KUKA KRL program: tipdress2.src, tipdress2.dat

--- tipdress2.src ---
&ACCESS RV1
&REL 33
&COMMENT TIPDRESS EXTERNAL GUN 2
DEF tipdress2( )
;================================================
; MODEL    :
; IE GROUP :
; STATION  :
; ROBOT    :
; FUNCTION : TIPDRESS EXTERNAL GUN 2
;================================================
;FOLD INI
;FOLD BASISTECH INI
GLOBAL INTERRUPT DECL 3 WHEN $STOPMESS==TRUE DO IR_STOPM ( )
INTERRUPT ON 3
BAS (#INITMOV,0 )
;ENDFOLD (BASISTECH INI)
;FOLD SPOTTECH INI
USERSPOT(#INIT)
;ENDFOLD (SPOTTECH INI)
;FOLD GRIPPERTECH INI
USER_GRP(0,DUMMY,DUMMY,GDEFAULT)
;ENDFOLD (GRIPPERTECH INI)
;FOLD USER INI
;Make your modifications here
;ENDFOLD (USER INI)
;ENDFOLD (INI)


pgno1_type=0

;FOLD PTP P10 H RETR OPN Gun= 2 Pair= FIRST Tool[14]:C520 Sin Pieza Base[0];%{PE}%R 6.1.2,%MKUKATPSPOT,%CRETR,%VPTP,%P 1:PTP, 2:P10, 3:, 5:100, 7:H, 9:#OPN, 11:2, 13:#FIRST
$BWDSTART=FALSE
PDAT_ACT=PH
FDAT_ACT=FP10
BAS(#PTP_PARAMS,PH.VEL)
S_ACT.GUN=2
S_ACT.PAIR=#FIRST
S_ACT.RETR=#OPN
S_READY=FALSE
TRIGGER WHEN DISTANCE=1 DELAY=0.0 DO USERSPOT(#RETR, S_ACT) PRIO=-1
PTP XP10
WAIT FOR S_READY
;ENDFOLD

;FOLD TDRESS.Swing_Forward 2 ;%{PE}%MKUKATPUSER
B_TDRESS=TDRESS (#SW_FWD ,2)
;ENDFOLD

;FOLD WAIT Time=1.5 sec;%{PE}%R 5.6.13,%MKUKATPBASIS,%CWAIT,%VWAIT,%P 2:1.5
WAIT SEC 1.5
;ENDFOLD

REPEAT

;FOLD TDRESS.Select_Active_Electrode 2 ;%{PE}%MKUKATPUSER
B_TDRESS=TDRESS (#TD_SEL ,2)
;ENDFOLD

pgno1_type=0
PGNO1=66

;FOLD TDRESS.Start_Cutter_Gun 2 ;%{PE}%MKUKATPUSER
B_TDRESS=TDRESS (#TD_START ,2)
;ENDFOLD

;FOLD TDRESS.Start_Count_Rotations 2 ;%{PE}%MKUKATPUSER
B_TDRESS=TDRESS (#CNT_STRT ,2)
;ENDFOLD

;FOLD CLOSE GUN 2 (3 TIMES) AND CHECK
$ADVANCE=0

FOR I=1 TO  3
CLOSEGUN (3 )

WAIT SEC 0.9



OPENGUN (3 )
ENDFOR
$ADVANCE=3
;endfold

;FOLD TDRESS.Stop_Count_Rotations 2 ;%{PE}%MKUKATPUSER
B_TDRESS=TDRESS (#CNT_STOP ,2)
;ENDFOLD

;FOLD TDRESS.Check_Rotations_Gun 2 Amount Of Rotations , 2 ;%{PE}%MKUKATPUSER
B_TDRESS=TDRESS (#CNT_CHK ,2, 2)
;ENDFOLD

UNTIL B_TDRESS==TRUE

;OPEN ARM OF THE DRESS

;FOLD TDRESS.Swing_Backward 2 ;%{PE}%MKUKATPUSER
B_TDRESS=TDRESS (#SW_BWD ,2)
;ENDFOLD

;FOLD TDRESS.Reset_Counter_Timer 2  Gun nr, 1 ;%{PE}%MKUKATPUSER
B_TDRESS=TDRESS (#TD_RES_CNT ,2, 1)
;ENDFOLD

;FOLD PTP Best_Praktisch H SPOT Gun= 2 Pair= FIRST RETR OPN INDEX1= 64 INDEX2= 1 Tool[14]:C520 Sin Pieza Base[0];%{PE}%R 6.1.2,%MKUKATPSPOT,%CSPOT,%VPTP,%P 1:PTP, 2:Best_Praktisch, 3:, 5:100, 7:H, 10:2, 12:#FIRST, 14:#OPN, 16:64, 18:1, 20:0, 22:0, 24:0, 25:SDAT3
$BWDSTART=FALSE
PDAT_ACT=PH
FDAT_ACT=FBest_Praktisch
BAS(#PTP_PARAMS,PH.VEL)
S_ACT.GUN=2
S_ACT.PAIR=#FIRST
S_ACT.RETR=#OPN
S_ACT.CLO_TM=SDEFAULT.CLO_TM
S_ACT.PGNO1=64
S_ACT.PGNO2=1
S_ACT.PRESS1=SDEFAULT.PRESS1
S_ACT.PRESS2=SDEFAULT.PRESS2
S_READY=FALSE
USERSPOT(#ADVSPOT, S_ACT)
TRIGGER WHEN DISTANCE=1 DELAY=SDEFAULT.CLO_TM DO USERSPOT(#PRESPOT, S_ACT) PRIO=-1
TRIGGER WHEN DISTANCE=1 DELAY=0.0 DO USERSPOT(#SPOT, S_ACT) PRIO=-1
PTP XBest_Praktisch
WAIT FOR S_READY
;ENDFOLD


END

;FOLD SETOUTPUT - SETS OUTPUT IF CONDITIONS ARE OK
DEF  SETOUTPUT (NR :IN,STATE :IN )
;************************************************************
;Function:  sets if to state value
;************************************************************
INT NR
BOOL STATE

IF (NR<>0) THEN
IF (NR>0) THEN
CONTINUE
$OUT[NR]=STATE
ELSE
CONTINUE
$OUT[-NR]= NOT STATE
ENDIF
ENDIF
END ;SetOutput
;ENDFOLD

;FOLD CHKINPUT - CHECKS INPUT <1 & RETURNS INPUT VALUE
DEFFCT  BOOL CHKINPUT(NR :IN,STATE :IN)
;************************************************************
;Function: checks if input nr<1 and returns input value
;************************************************************
INT NR
BOOL STATE

IF (NR<>0) THEN
IF (NR>0) THEN
RETURN  ($IN[NR]==STATE)
ELSE
RETURN  ($IN[-NR]==STATE)
ENDIF
ELSE
RETURN  (TRUE)
ENDIF
ENDFCT ; ChkInput
;ENDFOLD

;FOLD TIMEOUT - WAITS FOR CONDITION WITH TIMEOUT
DEFFCT  BOOL TIMEOUT(CONDITION :OUT,STATE :IN,MAXTIME :IN)
;************************************************************
;Function: waits for condition with timeout
;************************************************************
BOOL CONDITION
BOOL STATE
REAL MAXTIME

$TIMER[5]=-MAXTIME*1000
$TIMER_STOP[5]=FALSE
WHILE  (CONDITION<>STATE) AND  NOT ($TIMER_FLAG[5])
ENDWHILE
RETURN  ($TIMER_FLAG[5])
ENDFCT ; of TimeOut
;ENDFOLD

;FOLD CLOSEGUN - CLOSES WELDGUN BEFORE WELDING
DEF  CLOSEGUN (MYGUN :IN )
;************************************************************
;Function: closes and checks a gun
;************************************************************
INT MYGUN

SETOUTPUT (GRIPPER[MYGUN].OUT2,FALSE )
PULSE ($OUT[GRIPPER[MYGUN].OUT1],TRUE,0.2)
$TIMER[5]=-WAITTIME*1000
$TIMER_STOP[5]=FALSE
WHILE  ((CHKINPUT(GRIPPER[MYGUN].IN1,TRUE) AND CHKINPUT(GRIPPER[MYGUN].IN2,FALSE) AND CHKINPUT(GRIPPER[MYGUN].IN3,FALSE))<>TRUE) AND  NOT ($TIMER_FLAG[5])
ENDWHILE
IF ($TIMER_FLAG[5]) THEN
ERROR_DCP=TRUE
$MSG_T.RELEASE=FALSE
EMPTY_MSG={MSG_T: VALID FALSE,RELEASE FALSE,TYP #NOTIFY,MODUL[] " ",KEY[] " ",PARAM_TYP #VALUE,PARAM[] " ",DLG_FORMAT[] " ",ANSWER 0}
$MSG_T.TYP=#STATE
$MSG_T.KEY[]="Prestroke not closed        "
$MSG_T.VALID=TRUE
WAIT FOR  (($IN[GRIPPER[MYGUN].IN1]==TRUE) AND ($IN[GRIPPER[MYGUN].IN2]==FALSE) AND ($IN[GRIPPER[MYGUN].IN3]==FALSE))
$MSG_T.RELEASE=TRUE
WHILE $MSG_T.VALID
ENDWHILE
ERROR_DCP=FALSE
ENDIF

SETOUTPUT (GRIPPER[MYGUN].OUT3,TRUE )
SETOUTPUT (GRIPPER[MYGUN].OUT4,TRUE )
$TIMER[5]=-WAITTIME*1000
$TIMER_STOP[5]=FALSE
WHILE  ((CHKINPUT(GRIPPER[MYGUN].IN1,FALSE) AND CHKINPUT(GRIPPER[MYGUN].IN2,FALSE) AND CHKINPUT(GRIPPER[MYGUN].IN3,TRUE))<>TRUE) AND  NOT ($TIMER_FLAG[5])
ENDWHILE
IF ($TIMER_FLAG[5]) THEN
ERROR_DCP=TRUE
$MSG_T.RELEASE=FALSE
EMPTY_MSG={MSG_T: VALID FALSE,RELEASE FALSE,TYP #NOTIFY,MODUL[] " ",KEY[] " ",PARAM_TYP #VALUE,PARAM[] " ",DLG_FORMAT[] " ",ANSWER 0}
$MSG_T.TYP=#STATE
$MSG_T.KEY[]="Weldstroke not closed              "
$MSG_T.VALID=TRUE
WAIT FOR  (($IN[GRIPPER[MYGUN].IN1]==FALSE) AND ($IN[GRIPPER[MYGUN].IN2]==FALSE) AND ($IN[GRIPPER[MYGUN].IN3]==TRUE))
$MSG_T.RELEASE=TRUE
WHILE $MSG_T.VALID
ENDWHILE
ERROR_DCP=FALSE
ENDIF

END ;CLOSEGUN

;ENDFOLD

;FOLD OPENGUN - OPENS GUN FULLY AFTER WELDING
DEF  OPENGUN (MYGUN :IN )
;************************************************************
;Function: opens and checks a gun
;************************************************************
INT MYGUN
INT ANSWER

SETOUTPUT (GRIPPER[MYGUN].OUT3,FALSE )
SETOUTPUT (GRIPPER[MYGUN].OUT4,FALSE )
SETOUTPUT (GRIPPER[MYGUN].OUT1,FALSE )
PULSE ($OUT[GRIPPER[MYGUN].OUT2],TRUE,0.2)
$TIMER[5]=-WAITTIME*1000
$TIMER_STOP[5]=FALSE
WHILE  ((CHKINPUT(GRIPPER[MYGUN].IN1,FALSE) AND CHKINPUT(GRIPPER[MYGUN].IN2,TRUE) AND CHKINPUT(GRIPPER[MYGUN].IN3,FALSE))<>TRUE) AND  NOT ($TIMER_FLAG[5])
ENDWHILE
IF ($TIMER_FLAG[5]) THEN
ERROR_DCP=TRUE
$MSG_T.RELEASE=FALSE
EMPTY_MSG={MSG_T: VALID FALSE,RELEASE FALSE,TYP #NOTIFY,MODUL[] " ",KEY[] " ",PARAM_TYP #VALUE,PARAM[] " ",DLG_FORMAT[] " ",ANSWER 0}
$MSG_T.TYP=#STATE
$MSG_T.KEY[]="Prestroke not open                 "
$MSG_T.VALID=TRUE
WAIT FOR  (($IN[GRIPPER[MYGUN].IN1]==FALSE) AND ($IN[GRIPPER[MYGUN].IN2]==TRUE) AND ($IN[GRIPPER[MYGUN].IN3]==FALSE))
$MSG_T.RELEASE=TRUE
WHILE $MSG_T.VALID
ENDWHILE
ERROR_DCP=FALSE
ENDIF

END ;OPENGUN

--- tipdress2.dat ---
&ACCESS RV1
&REL 33
&COMMENT TIPDRESS EXTERNAL GUN 2
DEFDAT  TIPDRESS2
;FOLD EXTERNAL DECLARATIONS;%{PE}%MKUKATPBASIS,%CEXT,%VCOMMON,%P
;FOLD GRIPPERTECH EXT
EXT  H50 (INT  :IN,INT  :IN,INT  :IN,GRP_TYP  :IN )
;ENDFOLD (GRIPPERTECH EXT)
;FOLD SPOTTECH EXT
EXT  USERSPOT (S_COMMAND  :IN,SPOT_TYPE  :IN )
;ENDFOLD (SPOTTECH EXT)
;FOLD BASISTECH EXT;%{PE}%MKUKATPBASIS,%CEXT,%VEXT,%P
EXT  BAS (BAS_COMMAND  :IN,REAL  :IN )
DECL INT SUCCESS
;ENDFOLD (BASISTECH EXT)
;FOLD USER EXT;%{E}%MKUKATPUSER,%CEXT,%VEXT,%P
;Make here your modifications
;ENDFOLD (USER EXT)
;ENDFOLD (EXTERNAL DECLERATIONS)
;FOLD USER EXT;%{}%V2.2.2,%MKUKATPUSER,%CEXT,%VEXT,%P
;Make here your modifications
DECL BOOL TIPKONTROLE
DECL INT ANSWER
DECL INT WAITTIME=5
;ENDFOLD
;ENDFOLD
DECL INT I

;******************************
;*     E6POS Declarations     *
;******************************

DECL E6POS XP10={X 1812.73999,Y -758.109497,Z 1603.28101,A -10.9368095,B 87.2611084,C -2.35136199,S 6,T 50,E1 0.0,E2 0.0,E3 0.0,E4 0.0,E5 0.0,E6 0.0}
DECL E6POS XP20={X -1662.00305,Y -1200.49304,Z 238.679993,A 92.3594437,B 77.6989288,C -175.853195,S 6,T 26,E1 -667.745789,E2 0.0,E3 0.0,E4 0.0,E5 0.0,E6 0.0}
DECL E6POS XBEFORETIPDRESS={X -1664.84497,Y -1195.28101,Z 131.821106,A 92.7083206,B 79.2879791,C -177.241806,S 6,T 26,E1 -667.74939,E2 0.0,E3 0.0,E4 0.0,E5 0.0,E6 0.0}
DECL E6POS XDRESS_POS={X -1664.83301,Y -1250.33301,Z 131.817993,A 92.7068863,B 79.2882233,C -177.243393,S 6,T 26,E1 -667.74762,E2 0.0,E3 0.0,E4 0.0,E5 0.0,E6 0.0}
DECL E6POS XAFTERTIPDRESS={X -1664.84497,Y -1195.28101,Z 131.821106,A 92.7083206,B 79.2879791,C -177.241806,S 6,T 26,E1 -667.74939,E2 0.0,E3 0.0,E4 0.0,E5 0.0,E6 0.0}
DECL E6POS XBEST_PRACKTICE={X -1662.02905,Y -1184.83496,Z 277.771301,A 92.3578873,B 77.6946869,C -175.853302,S 6,T 26,E1 -667.74762,E2 0.0,E3 0.0,E4 0.0,E5 0.0,E6 0.0}
DECL E6POS XP30={X -958.122009,Y 929.273499,Z 985.610474,A 92.0788727,B 72.5539932,C -179.8358,S 6,T 26,E1 -2887.17505,E2 0.0,E3 0.0,E4 0.0,E5 0.0,E6 0.0}

;******************************
;*      FDAT Declarations     *
;******************************

DECL FDAT FP10={TOOL_NO 14,BASE_NO 0,IPO_FRAME #BASE,TQ_STATE FALSE}
DECL FDAT FP20={TOOL_NO 1,BASE_NO 0,IPO_FRAME #BASE}
DECL FDAT FBEFORETIPDRESS={TOOL_NO 1,BASE_NO 0,IPO_FRAME #BASE}
DECL FDAT FDRESS_POS={TOOL_NO 1,BASE_NO 0,IPO_FRAME #BASE}
DECL FDAT FAFTERTIPDRESS={TOOL_NO 1,BASE_NO 0,IPO_FRAME #BASE}
DECL FDAT FBEST_PRACKTICE={TOOL_NO 1,BASE_NO 0,IPO_FRAME #BASE}
DECL FDAT FP30={TOOL_NO 1,BASE_NO 0,IPO_FRAME #BASE}

;******************************
;*  PDAT & LDAT Declarations  *
;******************************

DECL PDAT PH={VEL 100.0,ACC 100.0,APO_DIST 100.0}

DECL E6POS XBEST_PRAKTISCH={X 1813.98499,Y -755.127197,Z 1603.28101,A -10.8495102,B 87.2611771,C -2.35826492,S 6,T 50,E1 0.0,E2 0.0,E3 0.0,E4 0.0,E5 0.0,E6 0.0}
DECL SPOT_SUGG_T LAST_SPOT={GUN[] "1                       ",RETR_CMD[] "#OPN                    ",CHOISE[] "#FIRST                  ",CLO_TM[] "0                       ",PGNO1[] "1                       ",PRESS1[] "0                       ",PGNO2[] "1                       ",PRESS2[] "0                       ",SPOT_PARAMS[] "SDAT3                   "}
DECL BASIS_SUGG_T LAST_BASIS={POINT1[] "Best_Praktisch          ",POINT2[] "Best_Praktisch          ",CP_PARAMS[] "CPDAT0                  ",PTP_PARAMS[] "H                       ",CONT[] "                        ",CP_VEL[] "2.0                     ",PTP_VEL[] "100                     ",SPL_NAME[] "S0                      "}
DECL FDAT FBest_Praktisch={TOOL_NO 14,BASE_NO 0,IPO_FRAME #BASE,POINT2[] " ",TQ_STATE FALSE}
DECL PDAT PPDAT1={VEL 100.0,ACC 100.0,APO_DIST 100.0}
DECL E6POS XBest_Praktice={X -1662.07202,Y -1184.76196,Z 277.795013,A 92.3631592,B 77.6921463,C -175.8461,S 6,T 26,E1 -667.74762,E2 0.0,E3 0.0,E4 0.0,E5 0.0,E6 0.0}
DECL FDAT FBest_Praktice={TOOL_NO 1,BASE_NO 0,IPO_FRAME #BASE,POINT2[] " "}
DECL E6POS XP21={X -929.55603,Y -159.533905,Z 748.283386,A 92.0804672,B 72.5703812,C -179.830597,S 6,T 26,E1 -2646.86792,E2 0.0,E3 0.0,E4 0.0,E5 0.0,E6 0.0}
DECL FDAT FP21={TOOL_NO 1,BASE_NO 0,IPO_FRAME #BASE}
DECL E6POS XP31={X -1185.09497,Y -662.41571,Z 415.422485,A 99.845192,B 75.8905869,C -168.599792,S 6,T 26,E1 -1294.38501,E2 0.0,E3 0.0,E4 0.0,E5 0.0,E6 0.0}
DECL FDAT FP31={TOOL_NO 1,BASE_NO 0,IPO_FRAME #BASE}
ENDDAT
